{attribute 'GeneratedUsingTerminal: EL9550-0010-0016'}
{attribute addProperty BoxType "EL9550-0010-0016"}
{attribute addProperty Id "EtcSlaveTerminalBaseStatus_UpAT %I*Status_Up_DB3531282Status_UsAT %I*Status_Us_DB3531282WcStateAT %I*WcState_9091E0EB2InfoDataAT %I*InfoData_6F19DB2B2"}
{attribute addProperty CRC "1491347839"}
{attribute addProperty Size "8"}
TYPE EL9550_58E4297F EXTENDS EtcSlaveTerminalBase :
STRUCT
	{attribute addProperty Name "Status_Up"}
	Status_Up : Status_Up_DB353128;
	{attribute addProperty Name "Status_Us"}
	Status_Us : Status_Us_DB353128;
	{attribute addProperty Name "WcState"}
	WcState : WcState_9091E0EB;
	{attribute addProperty Name "InfoData"}
	InfoData : InfoData_6F19DB2B;
END_STRUCT
END_TYPE

(* stored: Version 1.2.0.0, ProductVersion 3.1.4024.9
   DUT EL9550_58E4297F: Id {1d8d43cb-052f-42b0-8f2e-a57aa731bc6d} *)
